FUNCTION_BLOCK MQTT_STARTPOINT (* Peroidic event generator *)
  (* Standard: 61499-1 Annex A; Description: Copyright (c) 2017 fortiss GmbH This program and the accompanying materials are made available under the terms of the Eclipse Public License 2.0 which is available at https://www.eclipse.org/legal/epl-2.0/ SPDX-License-Identifier: EPL-2.0 *)
  (* Version 1.0, 2017-09-21, Alois Zoitl, fortiss GmbH, initial API and implementation and/or initial documentation *)
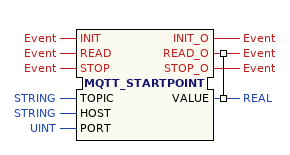
  EVENT_INPUT
    INIT;
    READ;
    STOP;
  END_EVENT
  EVENT_OUTPUT
    INIT_O;
    READ_O WITH VALUE;
    STOP_O;
  END_EVENT
  VAR_INPUT
    TOPIC : STRING; {SET_ATTRIBUTE(OpcUa, Constant)}
    HOST : STRING; {SET_ATTRIBUTE(OpcUa, Constant)}
    PORT : UINT; {SET_ATTRIBUTE(OpcUa, Constant)}
  END_VAR
  VAR_OUTPUT
    VALUE : REAL; {SET_ATTRIBUTE(OpcUa, Variable)}
  END_VAR
END_FUNCTION_BLOCK
(* other elements stored in the file *)
(* SelfDescription FBType=POINT.STARTPOINT *)
